FUNCTION_BLOCK App1_Pressure (* Composite Function Block Type *)
  (* Standard: 61499-2 *)
  (* Version 0.0, 2018-11-06, 4DIAC-IDE, 4DIAC-Consortium *)
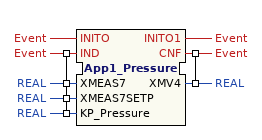
  EVENT_INPUT
    INITO; (* Initialization Request *)
    IND WITH XMEAS7, XMEAS7SETP, KP_Pressure; (* Normal Execution Request *)
  END_EVENT
  EVENT_OUTPUT
    INITO1; (* Initialization Confirm *)
    CNF WITH XMV4; (* Execution Confirmation *)
  END_EVENT
  VAR_INPUT
    XMEAS7 : REAL;
    XMEAS7SETP : REAL;
    KP_Pressure : REAL;
  END_VAR
  VAR_OUTPUT
    XMV4 : REAL;
  END_VAR
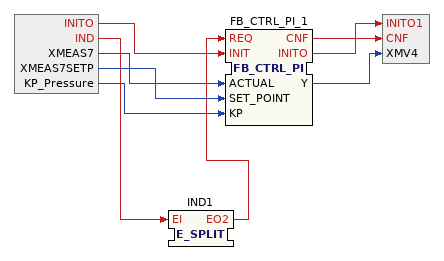
  FBS
    FB_CTRL_PI_1 : FB_CTRL_PI;
    IND1 : E_SPLIT;
  END_FBS
  EVENT_CONNECTIONS
    IND1.EO2 TO FB_CTRL_PI_1.REQ;
    IND TO IND1.EI;
    FB_CTRL_PI_1.CNF TO CNF;
    INITO TO FB_CTRL_PI_1.INIT;
    FB_CTRL_PI_1.INITO TO INITO1;
  END_CONNECTIONS
  DATA_CONNECTIONS
    XMEAS7 TO FB_CTRL_PI_1.ACTUAL;
    XMEAS7SETP TO FB_CTRL_PI_1.SET_POINT;
    FB_CTRL_PI_1.Y TO XMV4;
    KP_Pressure TO FB_CTRL_PI_1.KP;
  END_CONNECTIONS
END_FUNCTION_BLOCK
